// TIA Portal V17 export
// export: Created 2025-06-26T06:49:26.2112548Z, ExportSetting WithDefaults, DisplayName Totally Integrated Automation Portal, DisplayVersion V17 Update 8, DisplayName TIA Portal Openness, DisplayVersion V17 Update 8, DisplayName TIA Portal Version Control Interface, DisplayVersion V17, DisplayName STEP 7 Professional, DisplayVersion V17 Update 8, DisplayName STEP 7 Safety, DisplayVersion V17 Update 6, DisplayName WinCC Advanced, DisplayVersion V17 Update 8
DATA_BLOCK "DB_InverterDrives"   // DB41
{ S7_Optimized_Access := 'FALSE' }
AUTHOR : Heaten
VERSION : 0.1
// stored: AutoNumber true, DBAccessibleFromOPCUA true, DBAccessibleFromWebserver true, IsOnlyStoredInLoadMemory false, IsWriteProtectedInAS false
   VAR RETAIN
      CPC_SC_01 { S7_SetPoint := 'True'} : "stInverterDrive";   // CPC Cooling fan
      HBL_SC_01 { S7_SetPoint := 'True'} : "stInverterDrive";   // Container ventilation fan
      HBL_SC_02 { S7_SetPoint := 'True'} : "stInverterDrive";   // Compressor lubrication pump
      HBL_SC_03 { S7_SetPoint := 'True'} : "stInverterDrive";   // CPC Pump
      HBL_SC_10 { S7_SetPoint := 'True'} : "stInverterDrive";   // Compressor motor
   END_VAR
BEGIN
   CPC_SC_01.Cmd.Speed.Raw.iMax := 20000;
   CPC_SC_01.Cmd.Speed.Eng.fMax := 1500.0;
   CPC_SC_01.Cmd.Torque.Raw.iMax := 10000;
   CPC_SC_01.Cmd.Torque.Eng.fMax := 100.0;
   CPC_SC_01.Stat.Speed.Raw.iMax := 20000;
   CPC_SC_01.Stat.Speed.Eng.fMax := 1500.0;
   CPC_SC_01.Stat.Torque.Raw.iMax := 10000;
   CPC_SC_01.Stat.Torque.Eng.fMax := 100.0;
   CPC_SC_01.Stat.Power.Raw.iMax := 10000;
   CPC_SC_01.Stat.Power.Eng.fMax := 1.5;
   HBL_SC_01.Cmd.Speed.Raw.iMax := 20000;
   HBL_SC_01.Cmd.Speed.Eng.fMin := 0.0;
   HBL_SC_01.Cmd.Speed.Eng.fMax := 1500.0;
   HBL_SC_01.Cmd.Torque.Raw.iMax := 10000;
   HBL_SC_01.Cmd.Torque.Eng.fMax := 100.0;
   HBL_SC_01.Stat.Speed.Raw.iMax := 20000;
   HBL_SC_01.Stat.Speed.Eng.fMax := 1500.0;
   HBL_SC_01.Stat.Torque.Raw.iMax := 10000;
   HBL_SC_01.Stat.Torque.Eng.fMax := 100.0;
   HBL_SC_01.Stat.Power.Raw.iMax := 10000;
   HBL_SC_01.Stat.Power.Eng.fMax := 1.5;
   HBL_SC_02.Cmd.Speed.Raw.iMax := 20000;
   HBL_SC_02.Cmd.Speed.Eng.fMax := 5000.0;
   HBL_SC_02.Cmd.Torque.Raw.iMax := 10000;
   HBL_SC_02.Cmd.Torque.Eng.fMax := 100.0;
   HBL_SC_02.Stat.Speed.Raw.iMax := 20000;
   HBL_SC_02.Stat.Speed.Eng.fMax := 5000.0;
   HBL_SC_02.Stat.Torque.Raw.iMax := 10000;
   HBL_SC_02.Stat.Torque.Eng.fMax := 100.0;
   HBL_SC_02.Stat.Power.Raw.iMax := 10000;
   HBL_SC_02.Stat.Power.Eng.fMax := 2.0;
   HBL_SC_03.Cmd.Speed.Raw.iMax := 20000;
   HBL_SC_03.Cmd.Speed.Eng.fMax := 1500.0;
   HBL_SC_03.Cmd.Torque.Raw.iMax := 10000;
   HBL_SC_03.Cmd.Torque.Eng.fMax := 100.0;
   HBL_SC_03.Stat.Speed.Raw.iMax := 20000;
   HBL_SC_03.Stat.Speed.Eng.fMax := 1500.0;
   HBL_SC_03.Stat.Torque.Raw.iMax := 10000;
   HBL_SC_03.Stat.Torque.Eng.fMax := 100.0;
   HBL_SC_03.Stat.Power.Raw.iMax := 10000;
   HBL_SC_03.Stat.Power.Eng.fMax := 2.0;
   HBL_SC_10.Cmd.Speed.Raw.iMin := 0;
   HBL_SC_10.Cmd.Speed.Raw.iMax := 20000;
   HBL_SC_10.Cmd.Speed.Eng.fMin := 0.0;
   HBL_SC_10.Cmd.Speed.Eng.fMax := 1500.0;
   HBL_SC_10.Cmd.Torque.Raw.iMin := 0;
   HBL_SC_10.Cmd.Torque.Raw.iMax := 10000;
   HBL_SC_10.Cmd.Torque.Eng.fMin := 0.0;
   HBL_SC_10.Cmd.Torque.Eng.fMax := 100.0;
   HBL_SC_10.Stat.Speed.Raw.iMax := 20000;
   HBL_SC_10.Stat.Speed.Eng.fMin := 0.0;
   HBL_SC_10.Stat.Speed.Eng.fMax := 1500.0;
   HBL_SC_10.Stat.Torque.Raw.iMin := 0;
   HBL_SC_10.Stat.Torque.Raw.iMax := 10000;
   HBL_SC_10.Stat.Torque.Eng.fMin := 0.0;
   HBL_SC_10.Stat.Torque.Eng.fMax := 100.0;
   HBL_SC_10.Stat.Power.Raw.iMin := 0;
   HBL_SC_10.Stat.Power.Raw.iMax := 10000;
   HBL_SC_10.Stat.Power.Eng.fMin := 0.0;
   HBL_SC_10.Stat.Power.Eng.fMax := 1000.0;
END_DATA_BLOCK
